(* CoDeSys 2.3 export: MY.EXP *)

(* POU calc_time, CFC *)
FUNCTION_BLOCK calc_time
VAR_INPUT
	impuls: BOOL;
END_VAR
VAR_OUTPUT
	totalTime : UINT;
END_VAR
VAR
	rtirg1: R_TRIG;
	ton1: TON;
	res: BOOL;
	ftirg1: F_TRIG;
	tp1: TP;
	strt_ton: BOOL;
END_VAR
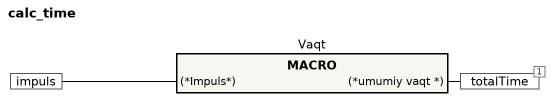
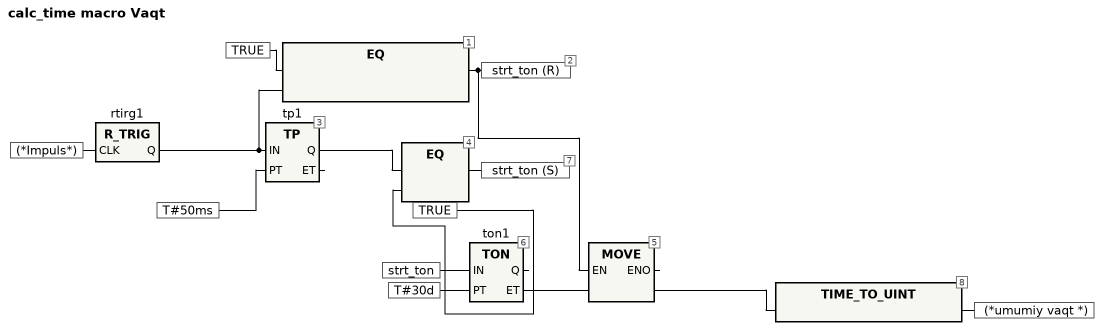
_CFC_ (* Continuous Function Chart, elements in execution order *)
#0 MACRO Vaqt(pin 1 "(*Impuls*)": impuls)
	#1 rtirg1:R_TRIG(CLK: pin 1)
	#2 EQ(TRUE, #1.Q)
	#3 R strt_ton <= #2
	#4 tp1:TP(IN: #1.Q, PT: T#50ms)
	#5 EQ(#4.Q, TRUE)
	#6 MOVE(EN: #2, #7.ET)
	#7 ton1:TON(IN: strt_ton, PT: T#30d)
	#8 S strt_ton <= #5
	out 1 "(*umumiy vaqt *)" <= #9
	#9 TIME_TO_UINT(#6)
END_MACRO
#10 totalTime <= #0.out 1
_END_CFC_
END_FUNCTION_BLOCK

(* POU CALCWEIGHT, CFC *)
FUNCTION_BLOCK CALCWEIGHT
VAR_INPUT
	milliVolt: REAL; 	(*Tenzo datchikdan keladigan millivolt*)
	dreyfNol: REAL; 	(*Tenzo datchikni usti bo'sh turgandagi millivolt*)
	koeffitsentPeredachaVes: REAL;	(*Koeffitsent peredacha ves na pogon metr*)
END_VAR
VAR_OUTPUT
	Ves: REAL;		(*Tenzo datchik o'lchgandan keyingi tayyor yuk kg da*)
END_VAR
VAR
END_VAR
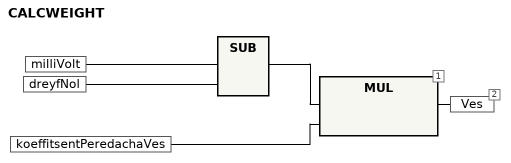
_CFC_ (* Continuous Function Chart, elements in execution order *)
#0 SUB(milliVolt, dreyfNol)
#1 MUL(#0, koeffitsentPeredachaVes)
#2 Ves <= #1
_END_CFC_
(* the same logic as Structured Text *)
Ves := (milliVolt - dreyfNol) * koeffitsentPeredachaVes;
END_FUNCTION_BLOCK

(* POU dozator, CFC *)
FUNCTION_BLOCK dozator
VAR_INPUT
	isIngroup: BOOL;		(*Dozator guruhda*)
	auto: BOOL;		(*Dozator avtomatik ishlamoqda*)
	koeffitsenPeredachVes : REAL;			(*Koeffitsent peredacha vesa*)

	length: REAL := 6.28;			 (*Impulslar orasidagi masofa*)
	impuls : BOOL;  				(*Sensordan kelayotgan impuls*)
	vaqt : DWORD := 3600;		 (* Impulsni makimal kutish vaqit*)
	reset_alarm: BOOL; 			(*Avariyani sboros qiqlish*)
END_VAR
VAR_OUTPUT
	zadaniyaChatotnika:REAL; (*CHastotnikka beriladigan volt yoki tok*)
END_VAR
VAR
	spd: speed;
END_VAR
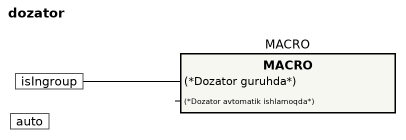
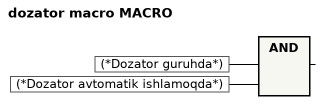
_CFC_ (* Continuous Function Chart, elements in execution order *)
#0 MACRO MACRO(pin 1 "(*Dozator guruhda*)": isIngroup, pin 2 "(*Dozator avtomatik ishlamoqda*)": -)
	#1 AND(pin 1, pin 2)
END_MACRO
unconnected input auto
_END_CFC_
END_FUNCTION_BLOCK

(* POU speed, CFC *)
FUNCTION_BLOCK speed
VAR_INPUT
	length: REAL := 6.28;			 (*Impulslar orasidagi masofa*)
	impuls : BOOL;  				(*Sensordan kelayotgan impuls*)
	vaqt : DWORD := 3600;		 (* Impulsni makimal kutish vaqit*)
	reset_alarm: BOOL; 				(*Avariyani sboros qiqlish*)
END_VAR
VAR_OUTPUT
	chastota : REAL; (*Kelayotgan impuls chastotasi*)
	tezlik : REAL; (*Impuls tezligi*)
	belt_alarm: BOOL; (* impulslar intervali "vaqt" dan oshib ketganda*)
END_VAR
VAR
	freq: FREQ_MEASURE;
	ton1: TON;
	calc_t: calc_time;
	ftrig3: F_TRIG;
	pere: BOOL;
	ton2: TON;
END_VAR
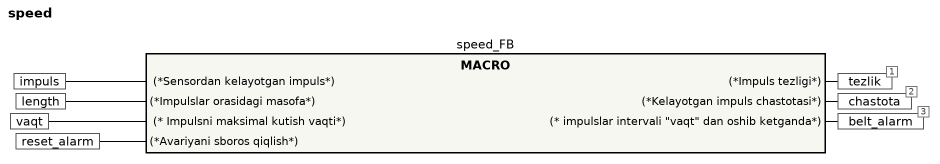
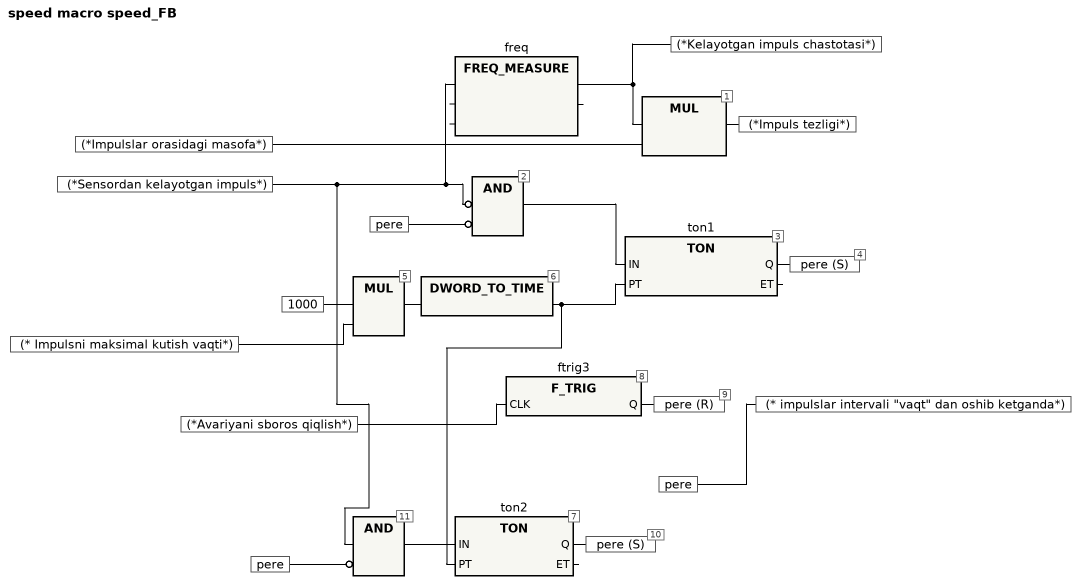
_CFC_ (* Continuous Function Chart, elements in execution order *)
#0 MACRO speed_FB(pin 1 "(*Sensordan kelayotgan impuls*)": impuls, pin 2 "(*Impulslar orasidagi masofa*)": length, pin 3 "(* Impulsni maksimal kutish vaqti*)": vaqt, pin 4 "(*Avariyani sboros qiqlish*)": reset_alarm)
	out 2 "(*Kelayotgan impuls chastotasi*)" <= #1.out 1
	#1 freq:FREQ_MEASURE(pin 1, -, -)
	#2 MUL(#1.out 1, pin 2)
	out 1 "(*Impuls tezligi*)" <= #2
	#3 AND(NOT pin 1, NOT pere)
	#4 ton1:TON(IN: #3, PT: #7)
	#5 S pere <= #4.Q
	#6 MUL(1000, pin 3)
	#7 DWORD_TO_TIME(#6)
	#8 ton2:TON(IN: #12, PT: #7)
	#9 ftrig3:F_TRIG(CLK: pin 4)
	#10 R pere <= #9.Q
	out 3 "(* impulslar intervali "vaqt" dan oshib ketganda*)" <= pere
	#11 S pere <= #8.Q
	#12 AND(pin 1, NOT pere)
END_MACRO
#13 tezlik <= #0.out 1
#14 chastota <= #0.out 2
#15 belt_alarm <= #0.out 3
_END_CFC_
END_FUNCTION_BLOCK

(* POU FILTRWEIGHT, CFC *)
FUNCTION_BLOCK FILTRWEIGHT
VAR_INPUT
	tmr1: TP;		(* Yukni filtrlash vaqti*)
	inputValue; 	(*Kiritilayotgan *)
END_VAR
VAR_OUTPUT
END_VAR
VAR

	rtig1: R_TRIG;

END_VAR
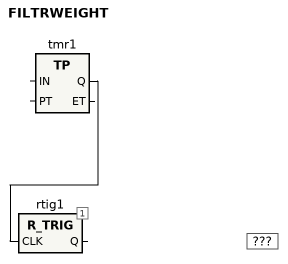
_CFC_ (* Continuous Function Chart, elements in execution order *)
#0 tmr1:TP(IN: -, PT: -)
#1 rtig1:R_TRIG(CLK: #0.Q)
unconnected input ???
_END_CFC_
(* the same logic as Structured Text *)
tmr1();
rtig1(CLK := tmr1.Q);
END_FUNCTION_BLOCK
